// TIA Portal V20 export
FUNCTION_BLOCK "CallGlobal"   // FB48, LAD
TITLE = CallGlobal
// All blocks that provide data to the DB Global.Data are called here. That includes blocks to generate system data as well as blocks that connect handle multiple HMIs.
// stored: IsIECCheckEnabled true, MemoryReserve 100, SetENOAutomatically true
   VAR
      statClockSysMemOld { ExternalWritable := 'False'} : Byte;   // Old value system memory evaluation
      statPulse : Array[0..9] of Bool;
      instLAF_PowerOnOff { ExternalWritable := 'False'} : "LAF_PowerOnOff";
      instLAF_HmiHeaderManager { ExternalWritable := 'False'} : "LAF_HmiHeaderManager";
      instLAF_ClockGen { ExternalWritable := 'False'} : "LAF_ClockGenerator";
      instLSNTP_Server { ExternalWritable := 'False'} : "LSNTP_Server";
      statTonTimer { ExternalWritable := 'False'} : Array[0..9] of TON_TIME;
   END_VAR
   VAR_TEMP
      tempIndex : DInt;   // Temp variable for for loop
      tempAcknowledge : Bool;   // Summarized acknowledge command
      tempPowerOff : Bool;   // Summarized power off command
      tempPowerOn : Bool;   // Summarized power on command
      tempPowerStatus : Int;   // 0 - Off, 1 - Paused, 2 - On
      tempResultXor : Byte;   // Interim result of XOR operation
      tempPosPulse : Byte;   // Interim result puls calculation
      temp_REPLACE_THIS : HW_ANY;
   END_VAR
   VAR CONSTANT
      RESET_BUTTON__COULD_BE_ADDED_HERE : Bool := false;   // Placeholder for a potential global reset button
      TRUE : Bool := TRUE;
      FALSE : Bool := FALSE;
   END_VAR
   VAR_TEMP   // added for the SCL form of the ladder/FBD networks
      _w1 : Bool;
      _w2 : Bool;
      _w3 : Bool;
      _w4 : Bool;
      _w5 : Bool;
      _w6 : Bool;
      _w7 : Bool;
      _w8 : Bool;
   END_VAR
BEGIN

REGION Network 1 (SCL): Summarize HMI commands
   // Read commands for acknowledge, powerOn and powerOff from the different HMI panels and summarize them in temp variables for further logic in this block.
   // Initialize temp variables
   #tempAcknowledge :=
   #tempPowerOff :=
   #tempPowerOn := FALSE;

   // Loop through the HMI panels and summarize the commands
   FOR #tempIndex := 0 TO "NO_OF_PANELS" DO
       #tempAcknowledge := #tempAcknowledge OR "Hmi".mainHeader[#tempIndex].hmiToPlc.acknowledge;
       #tempPowerOff := #tempPowerOff OR "Hmi".mainHeader[#tempIndex].hmiToPlc.powerCommands.%X0;
       #tempPowerOn := #tempPowerOn OR "Hmi".mainHeader[#tempIndex].hmiToPlc.powerCommands.%X1;
   END_FOR;
END_REGION

REGION Network 2: Global Acknowledge
   // The global acknowledge command from the hmi button is assigned to Global.Data.general.acknowledge: This bit it forwarded to all underlaying modules
   // If a hard-wired global reset button exists, it can
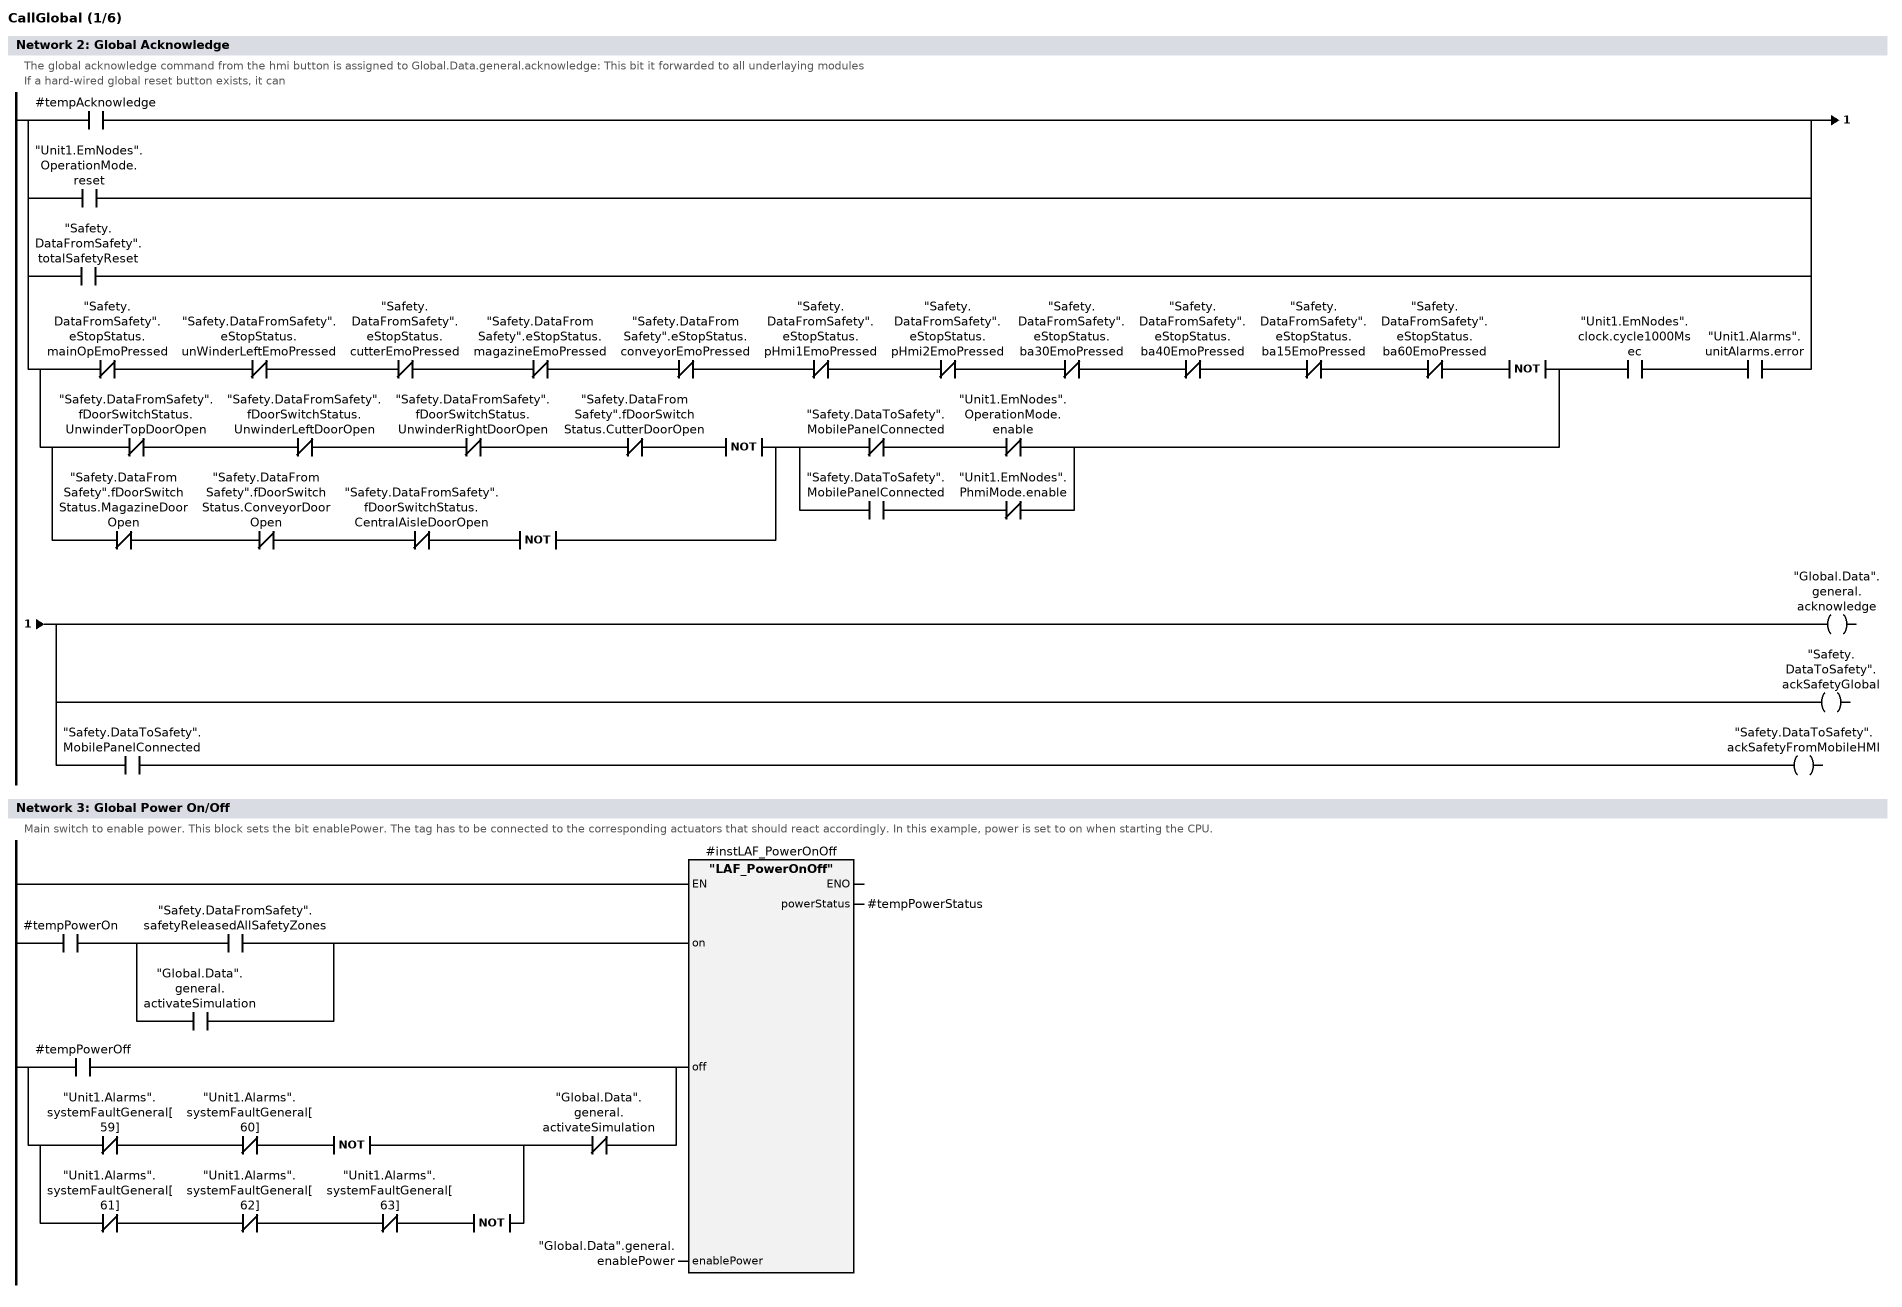
   RUNG wire#powerrail
      Contact( #tempAcknowledge )
      wire#w1
      Coil( "Global.Data".general.acknowledge )
   END_RUNG
   RUNG wire#powerrail
      Contact( "Unit1.EmNodes".OperationMode.reset )
   END_RUNG wire#w1
   RUNG wire#powerrail
      Contact( "Safety.DataFromSafety".totalSafetyReset )
   END_RUNG wire#w1
   RUNG wire#powerrail
      I_Contact( "Safety.DataFromSafety".eStopStatus.mainOpEmoPressed )
      I_Contact( "Safety.DataFromSafety".eStopStatus.unWinderLeftEmoPressed )
      I_Contact( "Safety.DataFromSafety".eStopStatus.cutterEmoPressed )
      I_Contact( "Safety.DataFromSafety".eStopStatus.magazineEmoPressed )
      I_Contact( "Safety.DataFromSafety".eStopStatus.conveyorEmoPressed )
      I_Contact( "Safety.DataFromSafety".eStopStatus.pHmi1EmoPressed )
      I_Contact( "Safety.DataFromSafety".eStopStatus.pHmi2EmoPressed )
      I_Contact( "Safety.DataFromSafety".eStopStatus.ba30EmoPressed )
      I_Contact( "Safety.DataFromSafety".eStopStatus.ba40EmoPressed )
      I_Contact( "Safety.DataFromSafety".eStopStatus.ba15EmoPressed )
      I_Contact( "Safety.DataFromSafety".eStopStatus.ba60EmoPressed )
      Not()
      wire#w2
      Contact( "Unit1.EmNodes".clock.cycle1000Msec )
      Contact( "Unit1.Alarms".unitAlarms.error )
   END_RUNG wire#w1
   RUNG wire#powerrail
      I_Contact( "Safety.DataFromSafety".fDoorSwitchStatus.UnwinderTopDoorOpen )
      I_Contact( "Safety.DataFromSafety".fDoorSwitchStatus.UnwinderLeftDoorOpen )
      I_Contact( "Safety.DataFromSafety".fDoorSwitchStatus.UnwinderRightDoorOpen )
      I_Contact( "Safety.DataFromSafety".fDoorSwitchStatus.CutterDoorOpen )
      Not()
      wire#w3
      I_Contact( "Safety.DataToSafety".MobilePanelConnected )
      I_Contact( "Unit1.EmNodes".OperationMode.enable )
   END_RUNG wire#w2
   RUNG wire#powerrail
      I_Contact( "Safety.DataFromSafety".fDoorSwitchStatus.MagazineDoorOpen )
      I_Contact( "Safety.DataFromSafety".fDoorSwitchStatus.ConveyorDoorOpen )
      I_Contact( "Safety.DataFromSafety".fDoorSwitchStatus.CentralAisleDoorOpen )
      Not()
   END_RUNG wire#w3
   RUNG wire#w3
      Contact( "Safety.DataToSafety".MobilePanelConnected )
      I_Contact( "Unit1.EmNodes".PhmiMode.enable )
   END_RUNG wire#w2
   RUNG wire#w1
      Coil( "Safety.DataToSafety".ackSafetyGlobal )
   END_RUNG
   RUNG wire#w1
      Contact( "Safety.DataToSafety".MobilePanelConnected )
      Coil( "Safety.DataToSafety".ackSafetyFromMobileHMI )
   END_RUNG
   // the same network as SCL:
   "Global.Data".general.acknowledge := #tempAcknowledge OR "Unit1.EmNodes".OperationMode.reset OR "Safety.DataFromSafety".totalSafetyReset OR ((NOT (NOT "Safety.DataFromSafety".eStopStatus.mainOpEmoPressed AND NOT "Safety.DataFromSafety".eStopStatus.unWinderLeftEmoPressed AND NOT "Safety.DataFromSafety".eStopStatus.cutterEmoPressed AND NOT "Safety.DataFromSafety".eStopStatus.magazineEmoPressed AND NOT "Safety.DataFromSafety".eStopStatus.conveyorEmoPressed AND NOT "Safety.DataFromSafety".eStopStatus.pHmi1EmoPressed AND NOT "Safety.DataFromSafety".eStopStatus.pHmi2EmoPressed AND NOT "Safety.DataFromSafety".eStopStatus.ba30EmoPressed AND NOT "Safety.DataFromSafety".eStopStatus.ba40EmoPressed AND NOT "Safety.DataFromSafety".eStopStatus.ba15EmoPressed AND NOT "Safety.DataFromSafety".eStopStatus.ba60EmoPressed) OR ((NOT (NOT "Safety.DataFromSafety".fDoorSwitchStatus.UnwinderTopDoorOpen AND NOT "Safety.DataFromSafety".fDoorSwitchStatus.UnwinderLeftDoorOpen AND NOT "Safety.DataFromSafety".fDoorSwitchStatus.UnwinderRightDoorOpen AND NOT "Safety.DataFromSafety".fDoorSwitchStatus.CutterDoorOpen) OR NOT (NOT "Safety.DataFromSafety".fDoorSwitchStatus.MagazineDoorOpen AND NOT "Safety.DataFromSafety".fDoorSwitchStatus.ConveyorDoorOpen AND NOT "Safety.DataFromSafety".fDoorSwitchStatus.CentralAisleDoorOpen)) AND ((NOT "Safety.DataToSafety".MobilePanelConnected AND NOT "Unit1.EmNodes".OperationMode.enable) OR ("Safety.DataToSafety".MobilePanelConnected AND NOT "Unit1.EmNodes".PhmiMode.enable)))) AND "Unit1.EmNodes".clock.cycle1000Msec AND "Unit1.Alarms".unitAlarms.error);
   "Safety.DataToSafety".ackSafetyGlobal := "Global.Data".general.acknowledge;
   "Safety.DataToSafety".ackSafetyFromMobileHMI := "Global.Data".general.acknowledge AND "Safety.DataToSafety".MobilePanelConnected;
END_REGION

REGION Network 3: Global Power On/Off
   // Main switch to enable power. This block sets the bit enablePower. The tag has to be connected to the corresponding actuators that should react accordingly. In this example, power is set to on when starting the CPU.
   RUNG wire#powerrail
      #instLAF_PowerOnOff(on := wire#w2, off := wire#w4, enablePower := "Global.Data".general.enablePower, powerStatus => #tempPowerStatus)
   END_RUNG
   RUNG wire#powerrail
      Contact( #tempPowerOn )
      wire#w1
      Contact( "Safety.DataFromSafety".safetyReleasedAllSafetyZones )
   END_RUNG wire#w2
   RUNG wire#w1
      Contact( "Global.Data".general.activateSimulation )
   END_RUNG wire#w2
   RUNG wire#powerrail
      Contact( #tempPowerOff )
   END_RUNG wire#w4
   RUNG wire#powerrail
      I_Contact( "Unit1.Alarms".systemFaultGeneral[59] )
      I_Contact( "Unit1.Alarms".systemFaultGeneral[60] )
      Not()
      wire#w3
      I_Contact( "Global.Data".general.activateSimulation )
   END_RUNG wire#w4
   RUNG wire#powerrail
      I_Contact( "Unit1.Alarms".systemFaultGeneral[61] )
      I_Contact( "Unit1.Alarms".systemFaultGeneral[62] )
      I_Contact( "Unit1.Alarms".systemFaultGeneral[63] )
      Not()
   END_RUNG wire#w3
   // the same network as SCL:
   #instLAF_PowerOnOff(on := #tempPowerOn AND ("Safety.DataFromSafety".safetyReleasedAllSafetyZones OR "Global.Data".general.activateSimulation),   // "LAF_PowerOnOff"
                       off := #tempPowerOff OR ((NOT (NOT "Unit1.Alarms".systemFaultGeneral[59] AND NOT "Unit1.Alarms".systemFaultGeneral[60]) OR NOT (NOT "Unit1.Alarms".systemFaultGeneral[61] AND NOT "Unit1.Alarms".systemFaultGeneral[62] AND NOT "Unit1.Alarms".systemFaultGeneral[63])) AND NOT "Global.Data".general.activateSimulation),
                       enablePower := "Global.Data".general.enablePower,
                       powerStatus => #tempPowerStatus);
END_REGION

REGION Network 4 (SCL): Write power status to HMI panels
   // Write power status back to all connected HMI panels
   // Loop through the panels and set the power status
   FOR #tempIndex := 0 TO "NO_OF_PANELS" DO
       "Hmi".mainHeader[#tempIndex].plcToHmi.powerStatus := #tempPowerStatus;
   END_FOR;
END_REGION

REGION Network 5: Special Function Buttons Operator Control Allowed
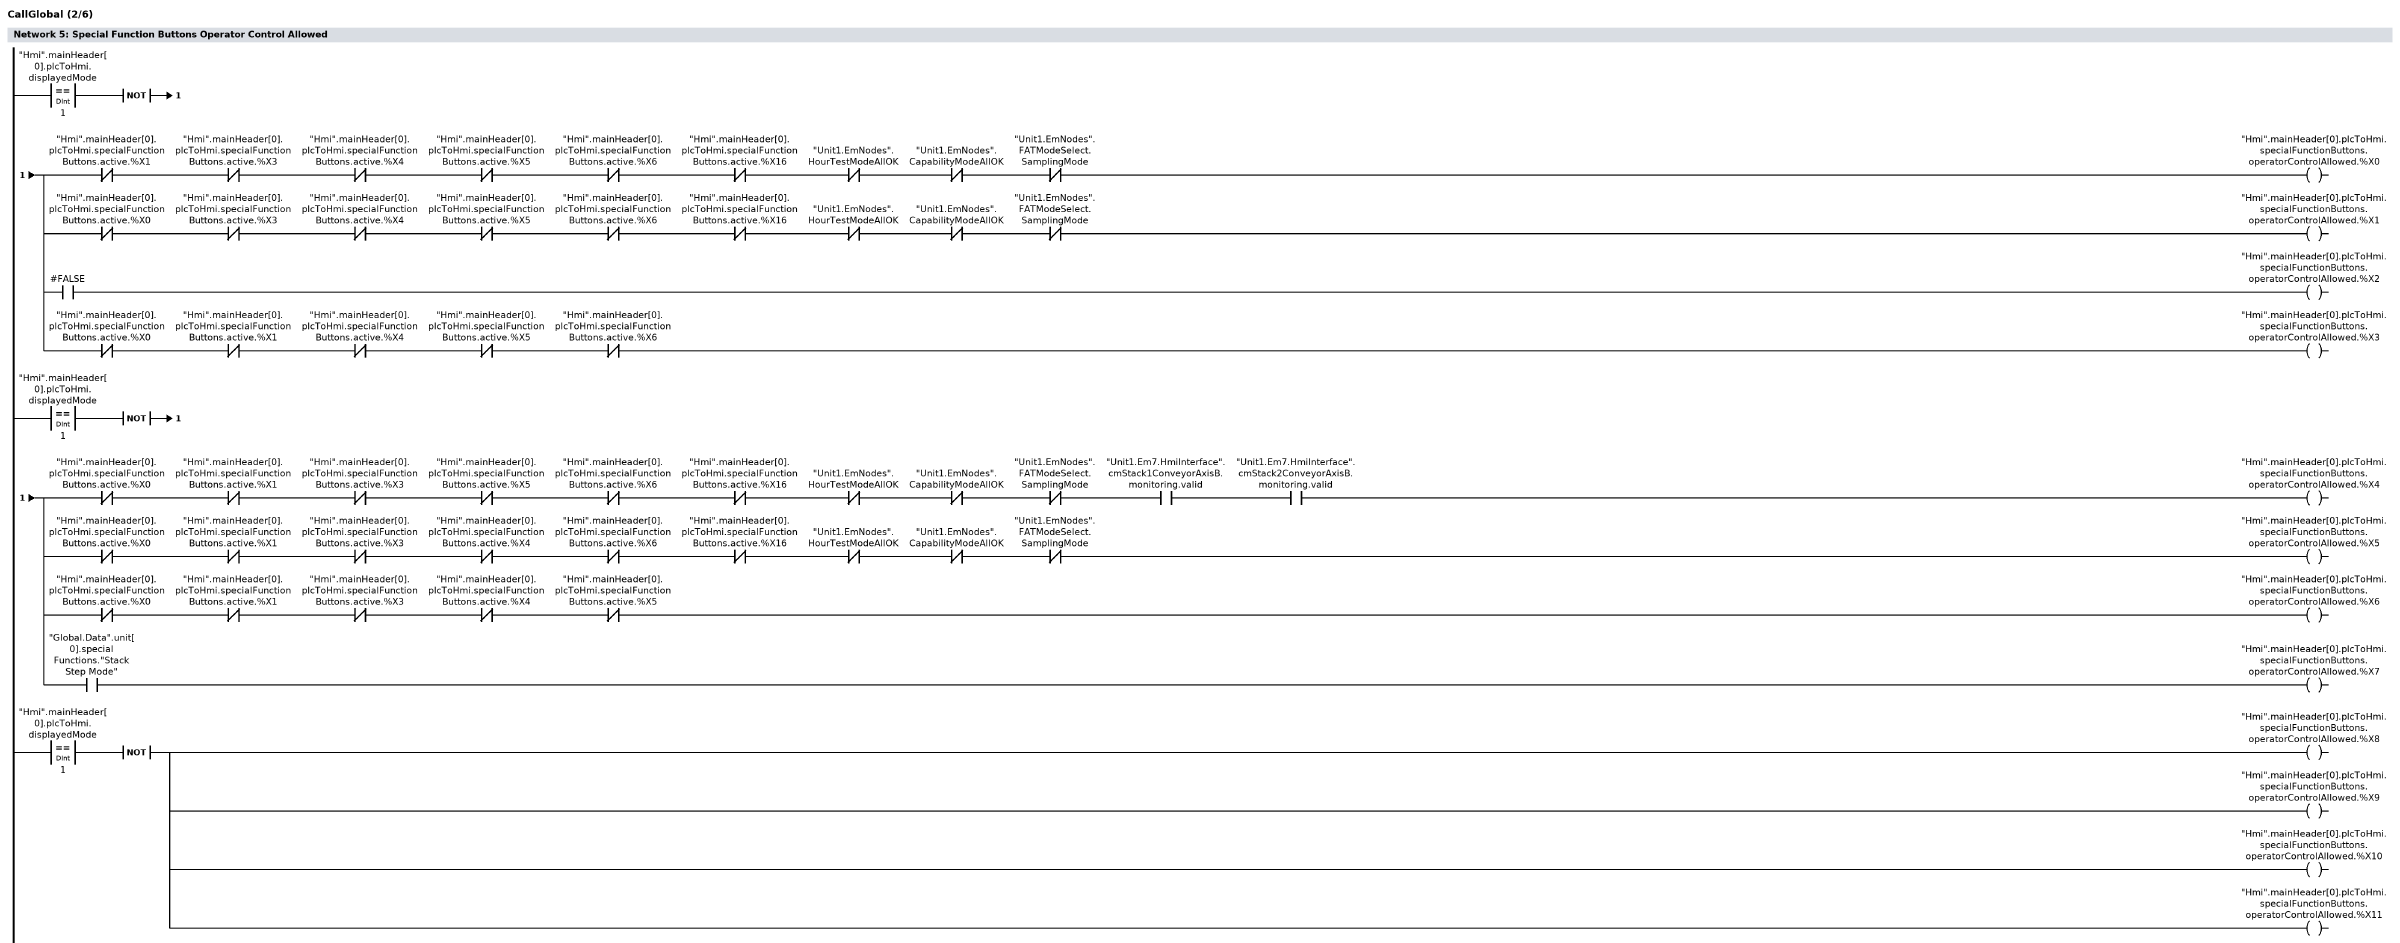
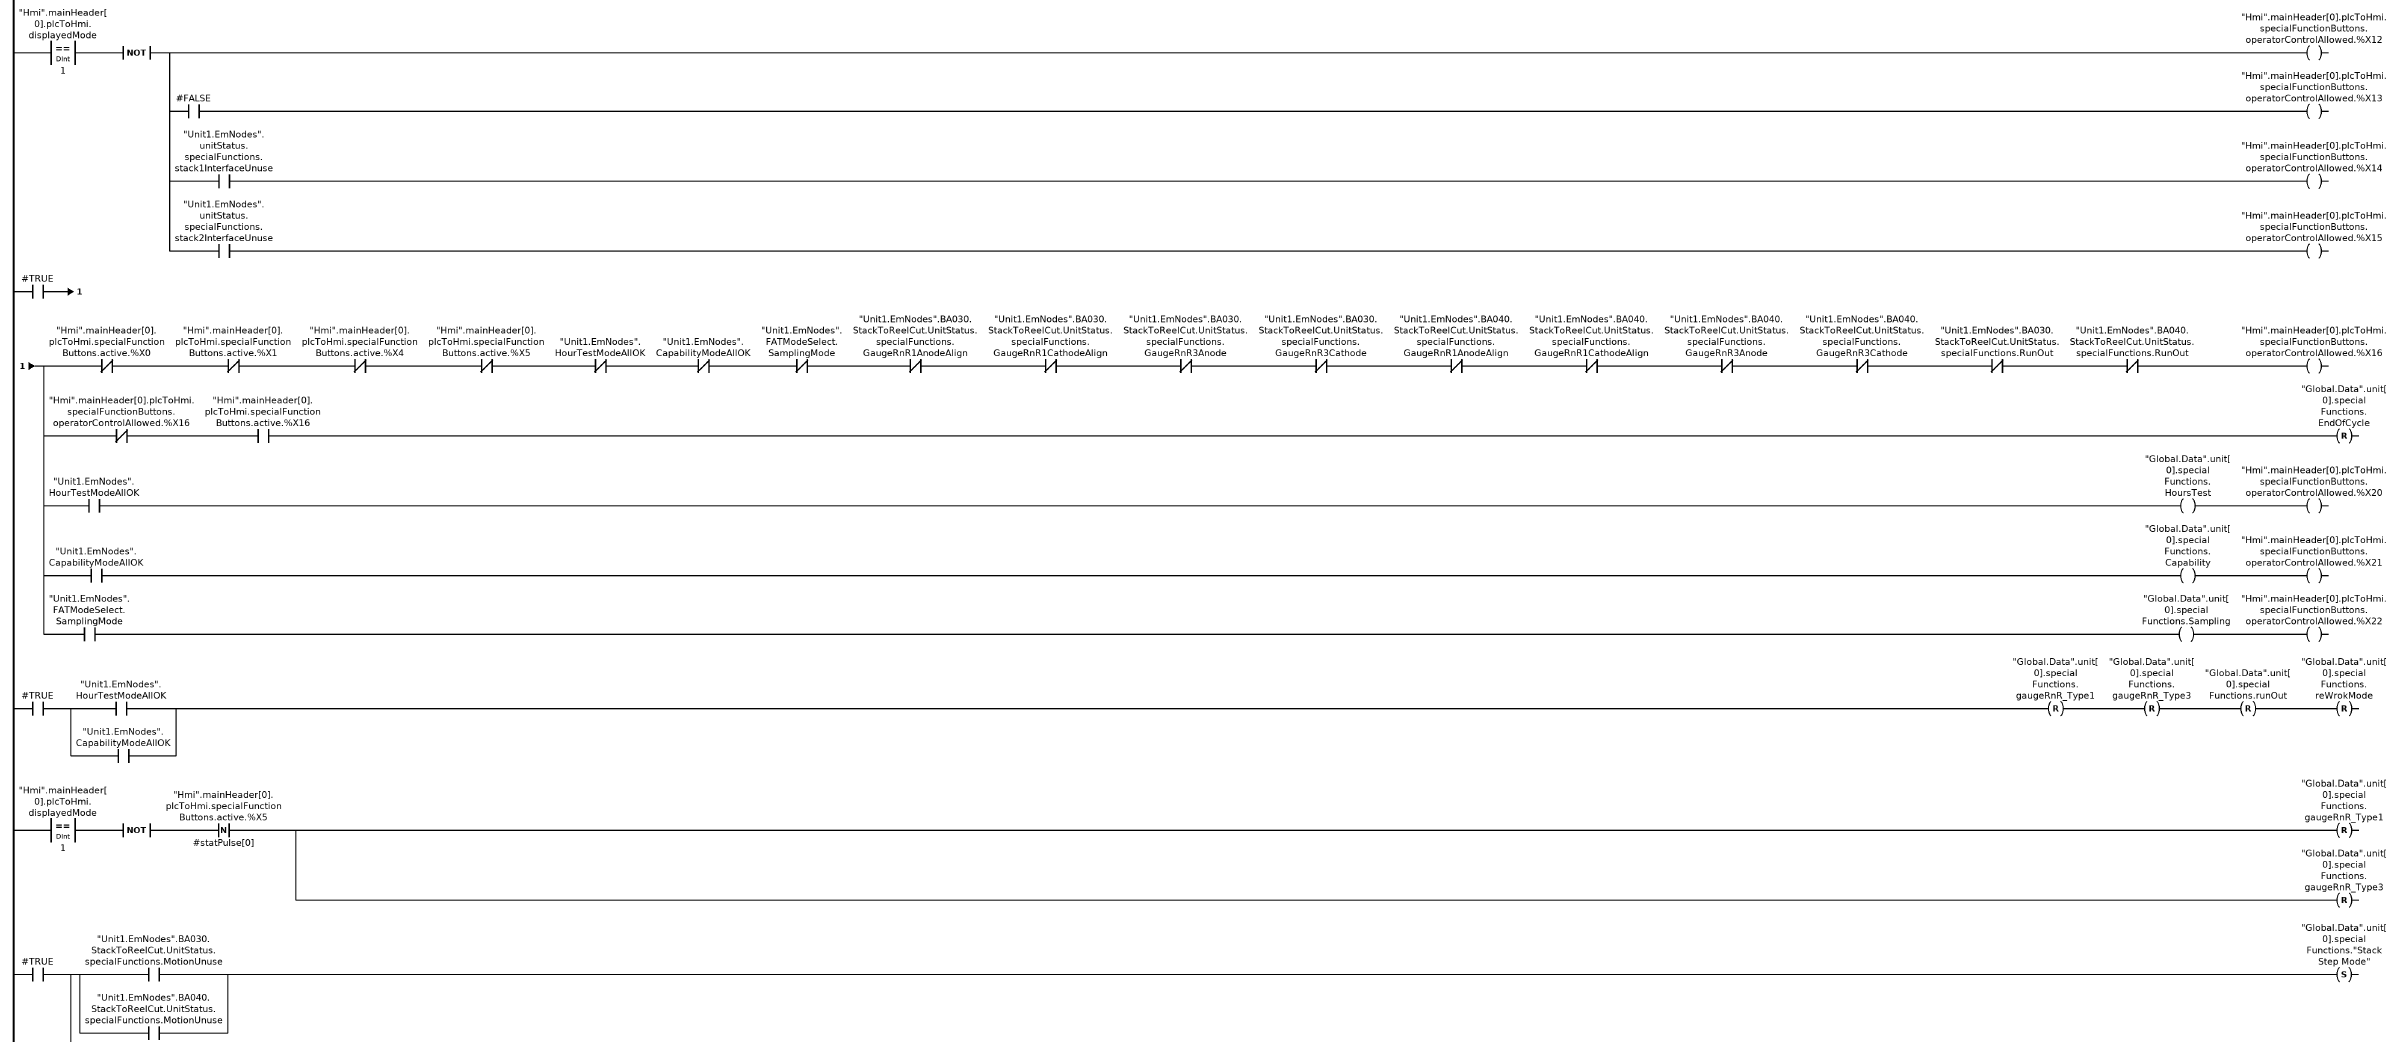
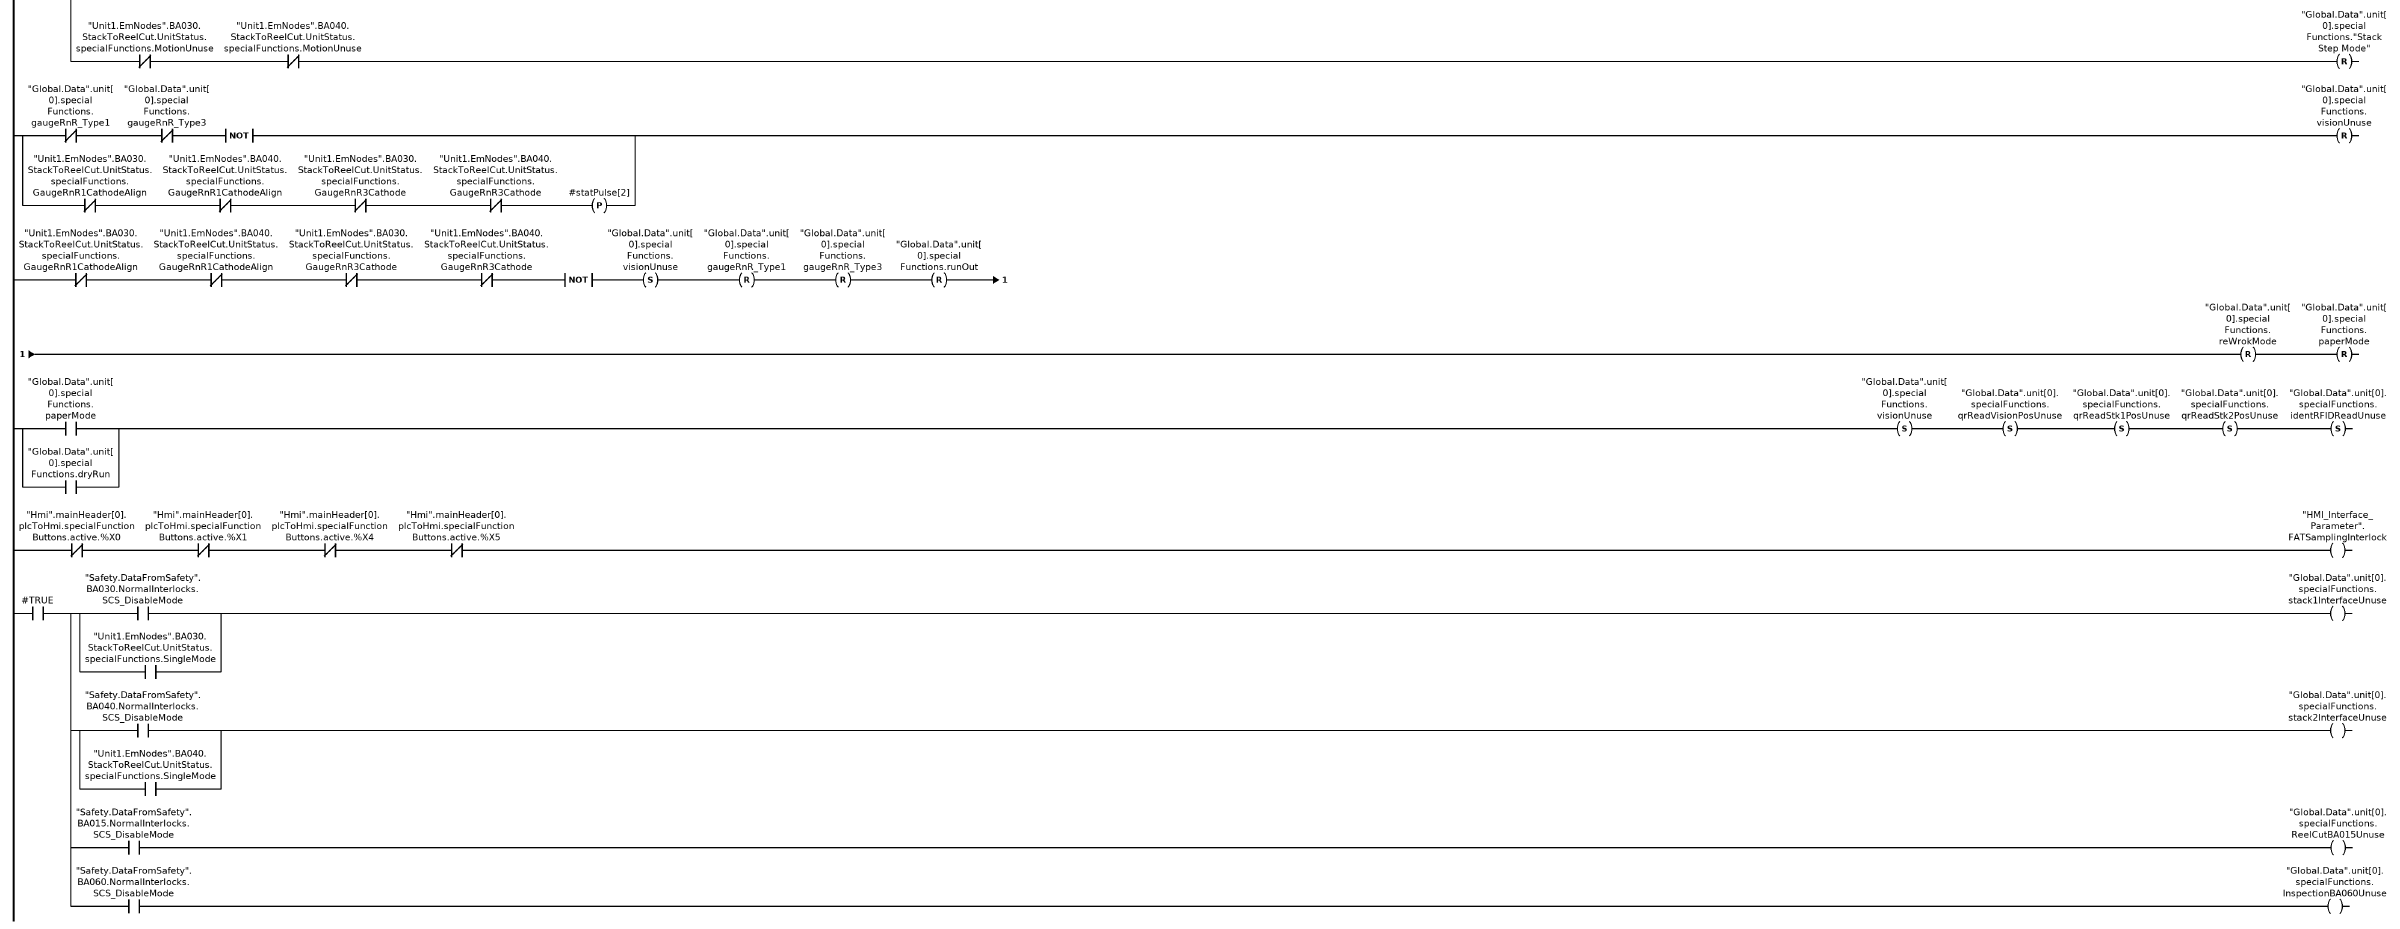
   RUNG wire#powerrail
      { S7_Templates := "SrcType := DInt" } EQ_Contact(in1 := "Hmi".mainHeader[0].plcToHmi.displayedMode, in2 := 1)
      Not()
      wire#w1
      I_Contact( "Hmi".mainHeader[0].plcToHmi.specialFunctionButtons.active.%X1 )
      I_Contact( "Hmi".mainHeader[0].plcToHmi.specialFunctionButtons.active.%X3 )
      I_Contact( "Hmi".mainHeader[0].plcToHmi.specialFunctionButtons.active.%X4 )
      I_Contact( "Hmi".mainHeader[0].plcToHmi.specialFunctionButtons.active.%X5 )
      I_Contact( "Hmi".mainHeader[0].plcToHmi.specialFunctionButtons.active.%X6 )
      I_Contact( "Hmi".mainHeader[0].plcToHmi.specialFunctionButtons.active.%X16 )
      I_Contact( "Unit1.EmNodes".HourTestModeAllOK )
      I_Contact( "Unit1.EmNodes".CapabilityModeAllOK )
      I_Contact( "Unit1.EmNodes".FATModeSelect.SamplingMode )
      Coil( "Hmi".mainHeader[0].plcToHmi.specialFunctionButtons.operatorControlAllowed.%X0 )
   END_RUNG
   RUNG wire#w1
      I_Contact( "Hmi".mainHeader[0].plcToHmi.specialFunctionButtons.active.%X0 )
      I_Contact( "Hmi".mainHeader[0].plcToHmi.specialFunctionButtons.active.%X3 )
      I_Contact( "Hmi".mainHeader[0].plcToHmi.specialFunctionButtons.active.%X4 )
      I_Contact( "Hmi".mainHeader[0].plcToHmi.specialFunctionButtons.active.%X5 )
      I_Contact( "Hmi".mainHeader[0].plcToHmi.specialFunctionButtons.active.%X6 )
      I_Contact( "Hmi".mainHeader[0].plcToHmi.specialFunctionButtons.active.%X16 )
      I_Contact( "Unit1.EmNodes".HourTestModeAllOK )
      I_Contact( "Unit1.EmNodes".CapabilityModeAllOK )
      I_Contact( "Unit1.EmNodes".FATModeSelect.SamplingMode )
      Coil( "Hmi".mainHeader[0].plcToHmi.specialFunctionButtons.operatorControlAllowed.%X1 )
   END_RUNG
   RUNG wire#w1
      Contact( #FALSE )
      Coil( "Hmi".mainHeader[0].plcToHmi.specialFunctionButtons.operatorControlAllowed.%X2 )
   END_RUNG
   RUNG wire#w1
      I_Contact( "Hmi".mainHeader[0].plcToHmi.specialFunctionButtons.active.%X0 )
      I_Contact( "Hmi".mainHeader[0].plcToHmi.specialFunctionButtons.active.%X1 )
      I_Contact( "Hmi".mainHeader[0].plcToHmi.specialFunctionButtons.active.%X4 )
      I_Contact( "Hmi".mainHeader[0].plcToHmi.specialFunctionButtons.active.%X5 )
      I_Contact( "Hmi".mainHeader[0].plcToHmi.specialFunctionButtons.active.%X6 )
      Coil( "Hmi".mainHeader[0].plcToHmi.specialFunctionButtons.operatorControlAllowed.%X3 )
   END_RUNG
   RUNG wire#powerrail
      { S7_Templates := "SrcType := DInt" } EQ_Contact(in1 := "Hmi".mainHeader[0].plcToHmi.displayedMode, in2 := 1)
      Not()
      wire#w2
      I_Contact( "Hmi".mainHeader[0].plcToHmi.specialFunctionButtons.active.%X0 )
      I_Contact( "Hmi".mainHeader[0].plcToHmi.specialFunctionButtons.active.%X1 )
      I_Contact( "Hmi".mainHeader[0].plcToHmi.specialFunctionButtons.active.%X3 )
      I_Contact( "Hmi".mainHeader[0].plcToHmi.specialFunctionButtons.active.%X5 )
      I_Contact( "Hmi".mainHeader[0].plcToHmi.specialFunctionButtons.active.%X6 )
      I_Contact( "Hmi".mainHeader[0].plcToHmi.specialFunctionButtons.active.%X16 )
      I_Contact( "Unit1.EmNodes".HourTestModeAllOK )
      I_Contact( "Unit1.EmNodes".CapabilityModeAllOK )
      I_Contact( "Unit1.EmNodes".FATModeSelect.SamplingMode )
      Contact( "Unit1.Em7.HmiInterface".cmStack1ConveyorAxisB.monitoring.valid )
      Contact( "Unit1.Em7.HmiInterface".cmStack2ConveyorAxisB.monitoring.valid )
      Coil( "Hmi".mainHeader[0].plcToHmi.specialFunctionButtons.operatorControlAllowed.%X4 )
   END_RUNG
   RUNG wire#w2
      I_Contact( "Hmi".mainHeader[0].plcToHmi.specialFunctionButtons.active.%X0 )
      I_Contact( "Hmi".mainHeader[0].plcToHmi.specialFunctionButtons.active.%X1 )
      I_Contact( "Hmi".mainHeader[0].plcToHmi.specialFunctionButtons.active.%X3 )
      I_Contact( "Hmi".mainHeader[0].plcToHmi.specialFunctionButtons.active.%X4 )
      I_Contact( "Hmi".mainHeader[0].plcToHmi.specialFunctionButtons.active.%X6 )
      I_Contact( "Hmi".mainHeader[0].plcToHmi.specialFunctionButtons.active.%X16 )
      I_Contact( "Unit1.EmNodes".HourTestModeAllOK )
      I_Contact( "Unit1.EmNodes".CapabilityModeAllOK )
      I_Contact( "Unit1.EmNodes".FATModeSelect.SamplingMode )
      Coil( "Hmi".mainHeader[0].plcToHmi.specialFunctionButtons.operatorControlAllowed.%X5 )
   END_RUNG
   RUNG wire#w2
      I_Contact( "Hmi".mainHeader[0].plcToHmi.specialFunctionButtons.active.%X0 )
      I_Contact( "Hmi".mainHeader[0].plcToHmi.specialFunctionButtons.active.%X1 )
      I_Contact( "Hmi".mainHeader[0].plcToHmi.specialFunctionButtons.active.%X3 )
      I_Contact( "Hmi".mainHeader[0].plcToHmi.specialFunctionButtons.active.%X4 )
      I_Contact( "Hmi".mainHeader[0].plcToHmi.specialFunctionButtons.active.%X5 )
      Coil( "Hmi".mainHeader[0].plcToHmi.specialFunctionButtons.operatorControlAllowed.%X6 )
   END_RUNG
   RUNG wire#w2
      Contact( "Global.Data".unit[0].specialFunctions."Stack Step Mode" )
      Coil( "Hmi".mainHeader[0].plcToHmi.specialFunctionButtons.operatorControlAllowed.%X7 )
   END_RUNG
   RUNG wire#powerrail
      { S7_Templates := "SrcType := DInt" } EQ_Contact(in1 := "Hmi".mainHeader[0].plcToHmi.displayedMode, in2 := 1)
      Not()
      wire#w3
      Coil( "Hmi".mainHeader[0].plcToHmi.specialFunctionButtons.operatorControlAllowed.%X8 )
   END_RUNG
   RUNG wire#w3
      Coil( "Hmi".mainHeader[0].plcToHmi.specialFunctionButtons.operatorControlAllowed.%X9 )
   END_RUNG
   RUNG wire#w3
      Coil( "Hmi".mainHeader[0].plcToHmi.specialFunctionButtons.operatorControlAllowed.%X10 )
   END_RUNG
   RUNG wire#w3
      Coil( "Hmi".mainHeader[0].plcToHmi.specialFunctionButtons.operatorControlAllowed.%X11 )
   END_RUNG
   RUNG wire#powerrail
      { S7_Templates := "SrcType := DInt" } EQ_Contact(in1 := "Hmi".mainHeader[0].plcToHmi.displayedMode, in2 := 1)
      Not()
      wire#w4
      Coil( "Hmi".mainHeader[0].plcToHmi.specialFunctionButtons.operatorControlAllowed.%X12 )
   END_RUNG
   RUNG wire#w4
      Contact( #FALSE )
      Coil( "Hmi".mainHeader[0].plcToHmi.specialFunctionButtons.operatorControlAllowed.%X13 )
   END_RUNG
   RUNG wire#w4
      Contact( "Unit1.EmNodes".unitStatus.specialFunctions.stack1InterfaceUnuse )
      Coil( "Hmi".mainHeader[0].plcToHmi.specialFunctionButtons.operatorControlAllowed.%X14 )
   END_RUNG
   RUNG wire#w4
      Contact( "Unit1.EmNodes".unitStatus.specialFunctions.stack2InterfaceUnuse )
      Coil( "Hmi".mainHeader[0].plcToHmi.specialFunctionButtons.operatorControlAllowed.%X15 )
   END_RUNG
   RUNG wire#powerrail
      Contact( #TRUE )
      wire#w5
      I_Contact( "Hmi".mainHeader[0].plcToHmi.specialFunctionButtons.active.%X0 )
      I_Contact( "Hmi".mainHeader[0].plcToHmi.specialFunctionButtons.active.%X1 )
      I_Contact( "Hmi".mainHeader[0].plcToHmi.specialFunctionButtons.active.%X4 )
      I_Contact( "Hmi".mainHeader[0].plcToHmi.specialFunctionButtons.active.%X5 )
      I_Contact( "Unit1.EmNodes".HourTestModeAllOK )
      I_Contact( "Unit1.EmNodes".CapabilityModeAllOK )
      I_Contact( "Unit1.EmNodes".FATModeSelect.SamplingMode )
      I_Contact( "Unit1.EmNodes".BA030.StackToReelCut.UnitStatus.specialFunctions.GaugeRnR1AnodeAlign )
      I_Contact( "Unit1.EmNodes".BA030.StackToReelCut.UnitStatus.specialFunctions.GaugeRnR1CathodeAlign )
      I_Contact( "Unit1.EmNodes".BA030.StackToReelCut.UnitStatus.specialFunctions.GaugeRnR3Anode )
      I_Contact( "Unit1.EmNodes".BA030.StackToReelCut.UnitStatus.specialFunctions.GaugeRnR3Cathode )
      I_Contact( "Unit1.EmNodes".BA040.StackToReelCut.UnitStatus.specialFunctions.GaugeRnR1AnodeAlign )
      I_Contact( "Unit1.EmNodes".BA040.StackToReelCut.UnitStatus.specialFunctions.GaugeRnR1CathodeAlign )
      I_Contact( "Unit1.EmNodes".BA040.StackToReelCut.UnitStatus.specialFunctions.GaugeRnR3Anode )
      I_Contact( "Unit1.EmNodes".BA040.StackToReelCut.UnitStatus.specialFunctions.GaugeRnR3Cathode )
      I_Contact( "Unit1.EmNodes".BA030.StackToReelCut.UnitStatus.specialFunctions.RunOut )
      I_Contact( "Unit1.EmNodes".BA040.StackToReelCut.UnitStatus.specialFunctions.RunOut )
      Coil( "Hmi".mainHeader[0].plcToHmi.specialFunctionButtons.operatorControlAllowed.%X16 )
   END_RUNG
   RUNG wire#w5
      I_Contact( "Hmi".mainHeader[0].plcToHmi.specialFunctionButtons.operatorControlAllowed.%X16 )
      Contact( "Hmi".mainHeader[0].plcToHmi.specialFunctionButtons.active.%X16 )
      R_Coil( "Global.Data".unit[0].specialFunctions.EndOfCycle )
   END_RUNG
   RUNG wire#w5
      Contact( "Unit1.EmNodes".HourTestModeAllOK )
      Coil( "Global.Data".unit[0].specialFunctions.HoursTest )
      Coil( "Hmi".mainHeader[0].plcToHmi.specialFunctionButtons.operatorControlAllowed.%X20 )
   END_RUNG
   RUNG wire#w5
      Contact( "Unit1.EmNodes".CapabilityModeAllOK )
      Coil( "Global.Data".unit[0].specialFunctions.Capability )
      Coil( "Hmi".mainHeader[0].plcToHmi.specialFunctionButtons.operatorControlAllowed.%X21 )
   END_RUNG
   RUNG wire#w5
      Contact( "Unit1.EmNodes".FATModeSelect.SamplingMode )
      Coil( "Global.Data".unit[0].specialFunctions.Sampling )
      Coil( "Hmi".mainHeader[0].plcToHmi.specialFunctionButtons.operatorControlAllowed.%X22 )
   END_RUNG
   RUNG wire#powerrail
      Contact( #TRUE )
      wire#w6
      Contact( "Unit1.EmNodes".HourTestModeAllOK )
      wire#w7
      R_Coil( "Global.Data".unit[0].specialFunctions.gaugeRnR_Type1 )
      R_Coil( "Global.Data".unit[0].specialFunctions.gaugeRnR_Type3 )
      R_Coil( "Global.Data".unit[0].specialFunctions.runOut )
      R_Coil( "Global.Data".unit[0].specialFunctions.reWrokMode )
   END_RUNG
   RUNG wire#w6
      Contact( "Unit1.EmNodes".CapabilityModeAllOK )
   END_RUNG wire#w7
   RUNG wire#powerrail
      { S7_Templates := "SrcType := DInt" } EQ_Contact(in1 := "Hmi".mainHeader[0].plcToHmi.displayedMode, in2 := 1)
      Not()
      N_Contact(operand := "Hmi".mainHeader[0].plcToHmi.specialFunctionButtons.active.%X5, bit := #statPulse[0])
      wire#w8
      R_Coil( "Global.Data".unit[0].specialFunctions.gaugeRnR_Type1 )
   END_RUNG
   RUNG wire#w8
      R_Coil( "Global.Data".unit[0].specialFunctions.gaugeRnR_Type3 )
   END_RUNG
   RUNG wire#powerrail
      Contact( #TRUE )
      wire#w9
      Contact( "Unit1.EmNodes".BA030.StackToReelCut.UnitStatus.specialFunctions.MotionUnuse )
      wire#w10
      S_Coil( "Global.Data".unit[0].specialFunctions."Stack Step Mode" )
   END_RUNG
   RUNG wire#w9
      Contact( "Unit1.EmNodes".BA040.StackToReelCut.UnitStatus.specialFunctions.MotionUnuse )
   END_RUNG wire#w10
   RUNG wire#w9
      I_Contact( "Unit1.EmNodes".BA030.StackToReelCut.UnitStatus.specialFunctions.MotionUnuse )
      I_Contact( "Unit1.EmNodes".BA040.StackToReelCut.UnitStatus.specialFunctions.MotionUnuse )
      R_Coil( "Global.Data".unit[0].specialFunctions."Stack Step Mode" )
   END_RUNG
   RUNG wire#powerrail
      I_Contact( "Global.Data".unit[0].specialFunctions.gaugeRnR_Type1 )
      I_Contact( "Global.Data".unit[0].specialFunctions.gaugeRnR_Type3 )
      Not()
      wire#w11
      R_Coil( "Global.Data".unit[0].specialFunctions.visionUnuse )
   END_RUNG
   RUNG wire#powerrail
      I_Contact( "Unit1.EmNodes".BA030.StackToReelCut.UnitStatus.specialFunctions.GaugeRnR1CathodeAlign )
      I_Contact( "Unit1.EmNodes".BA040.StackToReelCut.UnitStatus.specialFunctions.GaugeRnR1CathodeAlign )
      I_Contact( "Unit1.EmNodes".BA030.StackToReelCut.UnitStatus.specialFunctions.GaugeRnR3Cathode )
      I_Contact( "Unit1.EmNodes".BA040.StackToReelCut.UnitStatus.specialFunctions.GaugeRnR3Cathode )
      P_Trig( #statPulse[2] )
   END_RUNG wire#w11
   RUNG wire#powerrail
      I_Contact( "Unit1.EmNodes".BA030.StackToReelCut.UnitStatus.specialFunctions.GaugeRnR1CathodeAlign )
      I_Contact( "Unit1.EmNodes".BA040.StackToReelCut.UnitStatus.specialFunctions.GaugeRnR1CathodeAlign )
      I_Contact( "Unit1.EmNodes".BA030.StackToReelCut.UnitStatus.specialFunctions.GaugeRnR3Cathode )
      I_Contact( "Unit1.EmNodes".BA040.StackToReelCut.UnitStatus.specialFunctions.GaugeRnR3Cathode )
      Not()
      S_Coil( "Global.Data".unit[0].specialFunctions.visionUnuse )
      R_Coil( "Global.Data".unit[0].specialFunctions.gaugeRnR_Type1 )
      R_Coil( "Global.Data".unit[0].specialFunctions.gaugeRnR_Type3 )
      R_Coil( "Global.Data".unit[0].specialFunctions.runOut )
      R_Coil( "Global.Data".unit[0].specialFunctions.reWrokMode )
      R_Coil( "Global.Data".unit[0].specialFunctions.paperMode )
   END_RUNG
   RUNG wire#powerrail
      Contact( "Global.Data".unit[0].specialFunctions.paperMode )
      wire#w12
      S_Coil( "Global.Data".unit[0].specialFunctions.visionUnuse )
      S_Coil( "Global.Data".unit[0].specialFunctions.qrReadVisionPosUnuse )
      S_Coil( "Global.Data".unit[0].specialFunctions.qrReadStk1PosUnuse )
      S_Coil( "Global.Data".unit[0].specialFunctions.qrReadStk2PosUnuse )
      S_Coil( "Global.Data".unit[0].specialFunctions.identRFIDReadUnuse )
   END_RUNG
   RUNG wire#powerrail
      Contact( "Global.Data".unit[0].specialFunctions.dryRun )
   END_RUNG wire#w12
   RUNG wire#powerrail
      I_Contact( "Hmi".mainHeader[0].plcToHmi.specialFunctionButtons.active.%X0 )
      I_Contact( "Hmi".mainHeader[0].plcToHmi.specialFunctionButtons.active.%X1 )
      I_Contact( "Hmi".mainHeader[0].plcToHmi.specialFunctionButtons.active.%X4 )
      I_Contact( "Hmi".mainHeader[0].plcToHmi.specialFunctionButtons.active.%X5 )
      Coil( "HMI_Interface_Parameter".FATSamplingInterlock )
   END_RUNG
   RUNG wire#powerrail
      Contact( #TRUE )
      wire#w13
      Contact( "Safety.DataFromSafety".BA030.NormalInterlocks.SCS_DisableMode )
      wire#w14
      Coil( "Global.Data".unit[0].specialFunctions.stack1InterfaceUnuse )
   END_RUNG
   RUNG wire#w13
      Contact( "Unit1.EmNodes".BA030.StackToReelCut.UnitStatus.specialFunctions.SingleMode )
   END_RUNG wire#w14
   RUNG wire#w13
      Contact( "Safety.DataFromSafety".BA040.NormalInterlocks.SCS_DisableMode )
      wire#w15
      Coil( "Global.Data".unit[0].specialFunctions.stack2InterfaceUnuse )
   END_RUNG
   RUNG wire#w13
      Contact( "Unit1.EmNodes".BA040.StackToReelCut.UnitStatus.specialFunctions.SingleMode )
   END_RUNG wire#w15
   RUNG wire#w13
      Contact( "Safety.DataFromSafety".BA015.NormalInterlocks.SCS_DisableMode )
      Coil( "Global.Data".unit[0].specialFunctions.ReelCutBA015Unuse )
   END_RUNG
   RUNG wire#w13
      Contact( "Safety.DataFromSafety".BA060.NormalInterlocks.SCS_DisableMode )
      Coil( "Global.Data".unit[0].specialFunctions.InspectionBA060Unuse )
   END_RUNG
   // the same network as SCL:
   #_w1 := NOT ("Hmi".mainHeader[0].plcToHmi.displayedMode = 1);
   "Hmi".mainHeader[0].plcToHmi.specialFunctionButtons.operatorControlAllowed.%X0 := #_w1 AND NOT "Hmi".mainHeader[0].plcToHmi.specialFunctionButtons.active.%X1 AND NOT "Hmi".mainHeader[0].plcToHmi.specialFunctionButtons.active.%X3 AND NOT "Hmi".mainHeader[0].plcToHmi.specialFunctionButtons.active.%X4 AND NOT "Hmi".mainHeader[0].plcToHmi.specialFunctionButtons.active.%X5 AND NOT "Hmi".mainHeader[0].plcToHmi.specialFunctionButtons.active.%X6 AND NOT "Hmi".mainHeader[0].plcToHmi.specialFunctionButtons.active.%X16 AND NOT "Unit1.EmNodes".HourTestModeAllOK AND NOT "Unit1.EmNodes".CapabilityModeAllOK AND NOT "Unit1.EmNodes".FATModeSelect.SamplingMode;
   "Hmi".mainHeader[0].plcToHmi.specialFunctionButtons.operatorControlAllowed.%X1 := #_w1 AND NOT "Hmi".mainHeader[0].plcToHmi.specialFunctionButtons.active.%X0 AND NOT "Hmi".mainHeader[0].plcToHmi.specialFunctionButtons.active.%X3 AND NOT "Hmi".mainHeader[0].plcToHmi.specialFunctionButtons.active.%X4 AND NOT "Hmi".mainHeader[0].plcToHmi.specialFunctionButtons.active.%X5 AND NOT "Hmi".mainHeader[0].plcToHmi.specialFunctionButtons.active.%X6 AND NOT "Hmi".mainHeader[0].plcToHmi.specialFunctionButtons.active.%X16 AND NOT "Unit1.EmNodes".HourTestModeAllOK AND NOT "Unit1.EmNodes".CapabilityModeAllOK AND NOT "Unit1.EmNodes".FATModeSelect.SamplingMode;
   "Hmi".mainHeader[0].plcToHmi.specialFunctionButtons.operatorControlAllowed.%X2 := #_w1 AND #FALSE;
   "Hmi".mainHeader[0].plcToHmi.specialFunctionButtons.operatorControlAllowed.%X3 := #_w1 AND NOT "Hmi".mainHeader[0].plcToHmi.specialFunctionButtons.active.%X0 AND NOT "Hmi".mainHeader[0].plcToHmi.specialFunctionButtons.active.%X1 AND NOT "Hmi".mainHeader[0].plcToHmi.specialFunctionButtons.active.%X4 AND NOT "Hmi".mainHeader[0].plcToHmi.specialFunctionButtons.active.%X5 AND NOT "Hmi".mainHeader[0].plcToHmi.specialFunctionButtons.active.%X6;
   #_w2 := NOT ("Hmi".mainHeader[0].plcToHmi.displayedMode = 1);
   "Hmi".mainHeader[0].plcToHmi.specialFunctionButtons.operatorControlAllowed.%X4 := #_w2 AND NOT "Hmi".mainHeader[0].plcToHmi.specialFunctionButtons.active.%X0 AND NOT "Hmi".mainHeader[0].plcToHmi.specialFunctionButtons.active.%X1 AND NOT "Hmi".mainHeader[0].plcToHmi.specialFunctionButtons.active.%X3 AND NOT "Hmi".mainHeader[0].plcToHmi.specialFunctionButtons.active.%X5 AND NOT "Hmi".mainHeader[0].plcToHmi.specialFunctionButtons.active.%X6 AND NOT "Hmi".mainHeader[0].plcToHmi.specialFunctionButtons.active.%X16 AND NOT "Unit1.EmNodes".HourTestModeAllOK AND NOT "Unit1.EmNodes".CapabilityModeAllOK AND NOT "Unit1.EmNodes".FATModeSelect.SamplingMode AND "Unit1.Em7.HmiInterface".cmStack1ConveyorAxisB.monitoring.valid AND "Unit1.Em7.HmiInterface".cmStack2ConveyorAxisB.monitoring.valid;
   "Hmi".mainHeader[0].plcToHmi.specialFunctionButtons.operatorControlAllowed.%X5 := #_w2 AND NOT "Hmi".mainHeader[0].plcToHmi.specialFunctionButtons.active.%X0 AND NOT "Hmi".mainHeader[0].plcToHmi.specialFunctionButtons.active.%X1 AND NOT "Hmi".mainHeader[0].plcToHmi.specialFunctionButtons.active.%X3 AND NOT "Hmi".mainHeader[0].plcToHmi.specialFunctionButtons.active.%X4 AND NOT "Hmi".mainHeader[0].plcToHmi.specialFunctionButtons.active.%X6 AND NOT "Hmi".mainHeader[0].plcToHmi.specialFunctionButtons.active.%X16 AND NOT "Unit1.EmNodes".HourTestModeAllOK AND NOT "Unit1.EmNodes".CapabilityModeAllOK AND NOT "Unit1.EmNodes".FATModeSelect.SamplingMode;
   "Hmi".mainHeader[0].plcToHmi.specialFunctionButtons.operatorControlAllowed.%X6 := #_w2 AND NOT "Hmi".mainHeader[0].plcToHmi.specialFunctionButtons.active.%X0 AND NOT "Hmi".mainHeader[0].plcToHmi.specialFunctionButtons.active.%X1 AND NOT "Hmi".mainHeader[0].plcToHmi.specialFunctionButtons.active.%X3 AND NOT "Hmi".mainHeader[0].plcToHmi.specialFunctionButtons.active.%X4 AND NOT "Hmi".mainHeader[0].plcToHmi.specialFunctionButtons.active.%X5;
   "Hmi".mainHeader[0].plcToHmi.specialFunctionButtons.operatorControlAllowed.%X7 := #_w2 AND "Global.Data".unit[0].specialFunctions."Stack Step Mode";
   #_w3 := NOT ("Hmi".mainHeader[0].plcToHmi.displayedMode = 1);
   "Hmi".mainHeader[0].plcToHmi.specialFunctionButtons.operatorControlAllowed.%X8 := NOT ("Hmi".mainHeader[0].plcToHmi.displayedMode = 1);
   "Hmi".mainHeader[0].plcToHmi.specialFunctionButtons.operatorControlAllowed.%X9 := #_w3;
   "Hmi".mainHeader[0].plcToHmi.specialFunctionButtons.operatorControlAllowed.%X10 := #_w3;
   "Hmi".mainHeader[0].plcToHmi.specialFunctionButtons.operatorControlAllowed.%X11 := #_w3;
   #_w4 := NOT ("Hmi".mainHeader[0].plcToHmi.displayedMode = 1);
   "Hmi".mainHeader[0].plcToHmi.specialFunctionButtons.operatorControlAllowed.%X12 := NOT ("Hmi".mainHeader[0].plcToHmi.displayedMode = 1);
   "Hmi".mainHeader[0].plcToHmi.specialFunctionButtons.operatorControlAllowed.%X13 := #_w4 AND #FALSE;
   "Hmi".mainHeader[0].plcToHmi.specialFunctionButtons.operatorControlAllowed.%X14 := #_w4 AND "Unit1.EmNodes".unitStatus.specialFunctions.stack1InterfaceUnuse;
   "Hmi".mainHeader[0].plcToHmi.specialFunctionButtons.operatorControlAllowed.%X15 := #_w4 AND "Unit1.EmNodes".unitStatus.specialFunctions.stack2InterfaceUnuse;
   "Hmi".mainHeader[0].plcToHmi.specialFunctionButtons.operatorControlAllowed.%X16 := #TRUE AND NOT "Hmi".mainHeader[0].plcToHmi.specialFunctionButtons.active.%X0 AND NOT "Hmi".mainHeader[0].plcToHmi.specialFunctionButtons.active.%X1 AND NOT "Hmi".mainHeader[0].plcToHmi.specialFunctionButtons.active.%X4 AND NOT "Hmi".mainHeader[0].plcToHmi.specialFunctionButtons.active.%X5 AND NOT "Unit1.EmNodes".HourTestModeAllOK AND NOT "Unit1.EmNodes".CapabilityModeAllOK AND NOT "Unit1.EmNodes".FATModeSelect.SamplingMode AND NOT "Unit1.EmNodes".BA030.StackToReelCut.UnitStatus.specialFunctions.GaugeRnR1AnodeAlign AND NOT "Unit1.EmNodes".BA030.StackToReelCut.UnitStatus.specialFunctions.GaugeRnR1CathodeAlign AND NOT "Unit1.EmNodes".BA030.StackToReelCut.UnitStatus.specialFunctions.GaugeRnR3Anode AND NOT "Unit1.EmNodes".BA030.StackToReelCut.UnitStatus.specialFunctions.GaugeRnR3Cathode AND NOT "Unit1.EmNodes".BA040.StackToReelCut.UnitStatus.specialFunctions.GaugeRnR1AnodeAlign AND NOT "Unit1.EmNodes".BA040.StackToReelCut.UnitStatus.specialFunctions.GaugeRnR1CathodeAlign AND NOT "Unit1.EmNodes".BA040.StackToReelCut.UnitStatus.specialFunctions.GaugeRnR3Anode AND NOT "Unit1.EmNodes".BA040.StackToReelCut.UnitStatus.specialFunctions.GaugeRnR3Cathode AND NOT "Unit1.EmNodes".BA030.StackToReelCut.UnitStatus.specialFunctions.RunOut AND NOT "Unit1.EmNodes".BA040.StackToReelCut.UnitStatus.specialFunctions.RunOut;
   IF #TRUE AND NOT "Hmi".mainHeader[0].plcToHmi.specialFunctionButtons.operatorControlAllowed.%X16 AND "Hmi".mainHeader[0].plcToHmi.specialFunctionButtons.active.%X16 THEN
       "Global.Data".unit[0].specialFunctions.EndOfCycle := FALSE;
   END_IF;
   "Global.Data".unit[0].specialFunctions.HoursTest := #TRUE AND "Unit1.EmNodes".HourTestModeAllOK;
   "Hmi".mainHeader[0].plcToHmi.specialFunctionButtons.operatorControlAllowed.%X20 := #TRUE AND "Unit1.EmNodes".HourTestModeAllOK;
   "Global.Data".unit[0].specialFunctions.Capability := #TRUE AND "Unit1.EmNodes".CapabilityModeAllOK;
   "Hmi".mainHeader[0].plcToHmi.specialFunctionButtons.operatorControlAllowed.%X21 := #TRUE AND "Unit1.EmNodes".CapabilityModeAllOK;
   "Global.Data".unit[0].specialFunctions.Sampling := #TRUE AND "Unit1.EmNodes".FATModeSelect.SamplingMode;
   "Hmi".mainHeader[0].plcToHmi.specialFunctionButtons.operatorControlAllowed.%X22 := #TRUE AND "Unit1.EmNodes".FATModeSelect.SamplingMode;
   IF #TRUE AND ("Unit1.EmNodes".HourTestModeAllOK OR "Unit1.EmNodes".CapabilityModeAllOK) THEN
       "Global.Data".unit[0].specialFunctions.gaugeRnR_Type1 := FALSE;
       "Global.Data".unit[0].specialFunctions.gaugeRnR_Type3 := FALSE;
       "Global.Data".unit[0].specialFunctions.runOut := FALSE;
       "Global.Data".unit[0].specialFunctions.reWrokMode := FALSE;
   END_IF;
   #_w5 := NOT ("Hmi".mainHeader[0].plcToHmi.displayedMode = 1) AND NOT "Hmi".mainHeader[0].plcToHmi.specialFunctionButtons.active.%X5 AND #statPulse[0];   // falling edge of "Hmi".mainHeader[0].plcToHmi.specialFunctionButtons.active.%X5
   #statPulse[0] := "Hmi".mainHeader[0].plcToHmi.specialFunctionButtons.active.%X5;
   IF #_w5 THEN
       "Global.Data".unit[0].specialFunctions.gaugeRnR_Type1 := FALSE;
       "Global.Data".unit[0].specialFunctions.gaugeRnR_Type3 := FALSE;
   END_IF;
   IF #TRUE AND ("Unit1.EmNodes".BA030.StackToReelCut.UnitStatus.specialFunctions.MotionUnuse OR "Unit1.EmNodes".BA040.StackToReelCut.UnitStatus.specialFunctions.MotionUnuse) THEN
       "Global.Data".unit[0].specialFunctions."Stack Step Mode" := TRUE;
   END_IF;
   IF #TRUE AND NOT "Unit1.EmNodes".BA030.StackToReelCut.UnitStatus.specialFunctions.MotionUnuse AND NOT "Unit1.EmNodes".BA040.StackToReelCut.UnitStatus.specialFunctions.MotionUnuse THEN
       "Global.Data".unit[0].specialFunctions."Stack Step Mode" := FALSE;
   END_IF;
   #_w6 := NOT "Unit1.EmNodes".BA030.StackToReelCut.UnitStatus.specialFunctions.GaugeRnR1CathodeAlign AND NOT "Unit1.EmNodes".BA040.StackToReelCut.UnitStatus.specialFunctions.GaugeRnR1CathodeAlign AND NOT "Unit1.EmNodes".BA030.StackToReelCut.UnitStatus.specialFunctions.GaugeRnR3Cathode AND NOT "Unit1.EmNodes".BA040.StackToReelCut.UnitStatus.specialFunctions.GaugeRnR3Cathode;
   #_w7 := #_w6 AND NOT #statPulse[2];   // rising edge
   #statPulse[2] := #_w6;
   IF NOT (NOT "Global.Data".unit[0].specialFunctions.gaugeRnR_Type1 AND NOT "Global.Data".unit[0].specialFunctions.gaugeRnR_Type3) OR #_w7 THEN
       "Global.Data".unit[0].specialFunctions.visionUnuse := FALSE;
   END_IF;
   IF NOT (NOT "Unit1.EmNodes".BA030.StackToReelCut.UnitStatus.specialFunctions.GaugeRnR1CathodeAlign AND NOT "Unit1.EmNodes".BA040.StackToReelCut.UnitStatus.specialFunctions.GaugeRnR1CathodeAlign AND NOT "Unit1.EmNodes".BA030.StackToReelCut.UnitStatus.specialFunctions.GaugeRnR3Cathode AND NOT "Unit1.EmNodes".BA040.StackToReelCut.UnitStatus.specialFunctions.GaugeRnR3Cathode) THEN
       "Global.Data".unit[0].specialFunctions.visionUnuse := TRUE;
       "Global.Data".unit[0].specialFunctions.gaugeRnR_Type1 := FALSE;
       "Global.Data".unit[0].specialFunctions.gaugeRnR_Type3 := FALSE;
       "Global.Data".unit[0].specialFunctions.runOut := FALSE;
       "Global.Data".unit[0].specialFunctions.reWrokMode := FALSE;
       "Global.Data".unit[0].specialFunctions.paperMode := FALSE;
   END_IF;
   #_w8 := "Global.Data".unit[0].specialFunctions.paperMode OR "Global.Data".unit[0].specialFunctions.dryRun;
   IF #_w8 THEN
       "Global.Data".unit[0].specialFunctions.visionUnuse := TRUE;
       "Global.Data".unit[0].specialFunctions.qrReadVisionPosUnuse := TRUE;
       "Global.Data".unit[0].specialFunctions.qrReadStk1PosUnuse := TRUE;
       "Global.Data".unit[0].specialFunctions.qrReadStk2PosUnuse := TRUE;
       "Global.Data".unit[0].specialFunctions.identRFIDReadUnuse := TRUE;
   END_IF;
   "HMI_Interface_Parameter".FATSamplingInterlock := NOT "Hmi".mainHeader[0].plcToHmi.specialFunctionButtons.active.%X0 AND NOT "Hmi".mainHeader[0].plcToHmi.specialFunctionButtons.active.%X1 AND NOT "Hmi".mainHeader[0].plcToHmi.specialFunctionButtons.active.%X4 AND NOT "Hmi".mainHeader[0].plcToHmi.specialFunctionButtons.active.%X5;
   "Global.Data".unit[0].specialFunctions.stack1InterfaceUnuse := #TRUE AND ("Safety.DataFromSafety".BA030.NormalInterlocks.SCS_DisableMode OR "Unit1.EmNodes".BA030.StackToReelCut.UnitStatus.specialFunctions.SingleMode);
   "Global.Data".unit[0].specialFunctions.stack2InterfaceUnuse := #TRUE AND ("Safety.DataFromSafety".BA040.NormalInterlocks.SCS_DisableMode OR "Unit1.EmNodes".BA040.StackToReelCut.UnitStatus.specialFunctions.SingleMode);
   "Global.Data".unit[0].specialFunctions.ReelCutBA015Unuse := #TRUE AND "Safety.DataFromSafety".BA015.NormalInterlocks.SCS_DisableMode;
   "Global.Data".unit[0].specialFunctions.InspectionBA060Unuse := #TRUE AND "Safety.DataFromSafety".BA060.NormalInterlocks.SCS_DisableMode;
END_REGION

REGION Network 6: HMI Control Header
   // Read the input from the control header in the HMI an distribute information to the according units. Vice versa, summarize the unit information and provide it to the control header to display e.g. the modes and states.
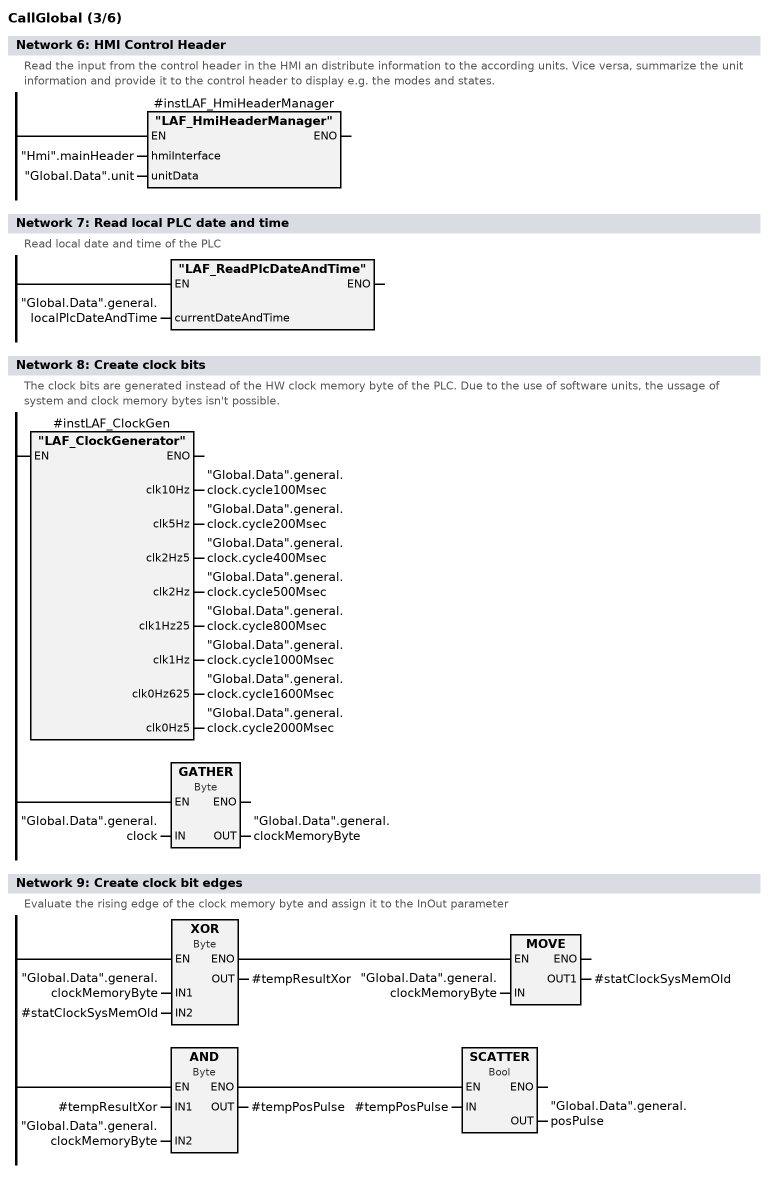
   RUNG wire#powerrail
      #instLAF_HmiHeaderManager(hmiInterface := "Hmi".mainHeader, unitData := "Global.Data".unit)
   END_RUNG
   // the same network as SCL:
   #instLAF_HmiHeaderManager(hmiInterface := "Hmi".mainHeader, unitData := "Global.Data".unit);   // "LAF_HmiHeaderManager"
END_REGION

REGION Network 7: Read local PLC date and time
   // Read local date and time of the PLC
   RUNG wire#powerrail
      "LAF_ReadPlcDateAndTime"(currentDateAndTime := "Global.Data".general.localPlcDateAndTime)
   END_RUNG
   // the same network as SCL:
   "LAF_ReadPlcDateAndTime"(currentDateAndTime := "Global.Data".general.localPlcDateAndTime);
END_REGION

REGION Network 8: Create clock bits
   // The clock bits are generated instead of the HW clock memory byte of the PLC. Due to the use of software units, the ussage of system and clock memory bytes isn't possible.
   RUNG wire#powerrail
      #instLAF_ClockGen(clk10Hz => "Global.Data".general.clock.cycle100Msec, clk5Hz => "Global.Data".general.clock.cycle200Msec, clk2Hz5 => "Global.Data".general.clock.cycle400Msec, clk2Hz => "Global.Data".general.clock.cycle500Msec, clk1Hz25 => "Global.Data".general.clock.cycle800Msec, clk1Hz => "Global.Data".general.clock.cycle1000Msec, clk0Hz625 => "Global.Data".general.clock.cycle1600Msec, clk0Hz5 => "Global.Data".general.clock.cycle2000Msec)
   END_RUNG
   RUNG wire#powerrail
      { S7_Templates := "[dest_type := Byte, src_type := Bool]" } GATHER(IN := "Global.Data".general.clock, OUT => "Global.Data".general.clockMemoryByte)
   END_RUNG
   // the same network as SCL:
   #instLAF_ClockGen(clk10Hz => "Global.Data".general.clock.cycle100Msec,   // "LAF_ClockGenerator"
                     clk5Hz => "Global.Data".general.clock.cycle200Msec,
                     clk2Hz5 => "Global.Data".general.clock.cycle400Msec,
                     clk2Hz => "Global.Data".general.clock.cycle500Msec,
                     clk1Hz25 => "Global.Data".general.clock.cycle800Msec,
                     clk1Hz => "Global.Data".general.clock.cycle1000Msec,
                     clk0Hz625 => "Global.Data".general.clock.cycle1600Msec,
                     clk0Hz5 => "Global.Data".general.clock.cycle2000Msec);
   GATHER(IN := "Global.Data".general.clock, OUT => "Global.Data".general.clockMemoryByte);
END_REGION

REGION Network 9: Create clock bit edges
   // Evaluate the rising edge of the clock memory byte and assign it to the InOut parameter
   #tempResultXor := "Global.Data".general.clockMemoryByte XOR #statClockSysMemOld;
   #statClockSysMemOld := "Global.Data".general.clockMemoryByte;
   #tempPosPulse := #tempResultXor AND "Global.Data".general.clockMemoryByte;
   SCATTER(IN := #tempPosPulse, OUT => "Global.Data".general.posPulse);
END_REGION

REGION Network 10: Time Synchronisation (NTP)
   // With the LSNTP_Server block, the NTP server will be enabled on S7 PLC, to wich the NTP client (e.g. Panel), can synchronize their data and time.
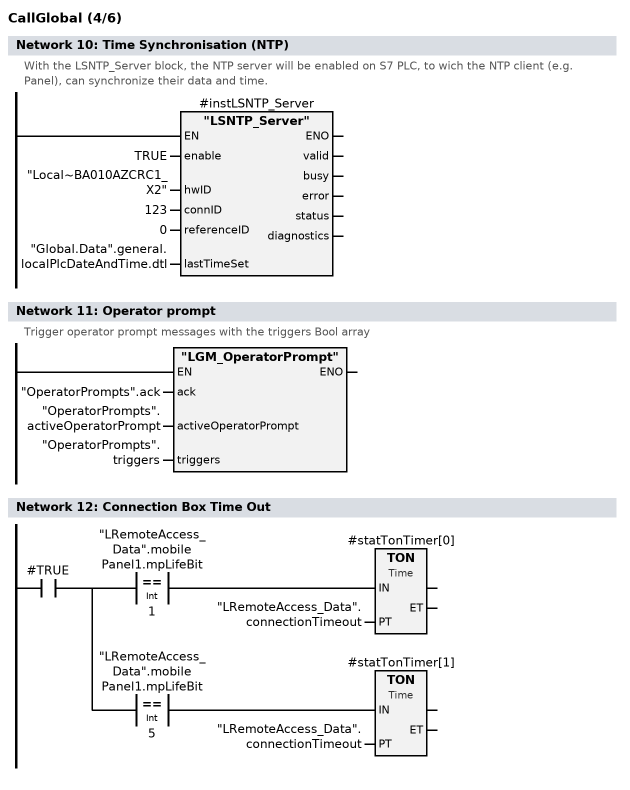
   RUNG wire#powerrail
      #instLSNTP_Server(enable := TRUE, hwID := "Local~BA010AZCRC1_X2", connID := 123, referenceID := 0, lastTimeSet := "Global.Data".general.localPlcDateAndTime.dtl, valid =>, busy =>, error =>, status =>, diagnostics =>)
   END_RUNG
   // the same network as SCL:
   #instLSNTP_Server(enable := TRUE,   // "LSNTP_Server"
                     hwID := "Local~BA010AZCRC1_X2",
                     connID := 123,
                     referenceID := 0,
                     lastTimeSet := "Global.Data".general.localPlcDateAndTime.dtl);
END_REGION

REGION Network 11: Operator prompt
   // Trigger operator prompt messages with the triggers Bool array
   RUNG wire#powerrail
      "LGM_OperatorPrompt"(ack := "OperatorPrompts".ack, activeOperatorPrompt := "OperatorPrompts".activeOperatorPrompt, triggers := "OperatorPrompts".triggers)
   END_RUNG
   // the same network as SCL:
   "LGM_OperatorPrompt"(ack := "OperatorPrompts".ack,
                        activeOperatorPrompt := "OperatorPrompts".activeOperatorPrompt,
                        triggers := "OperatorPrompts".triggers);
END_REGION

REGION Network 12: Connection Box Time Out
   RUNG wire#powerrail
      Contact( #TRUE )
      wire#w1
      { S7_Templates := "SrcType := Int" } EQ_Contact(in1 := "LRemoteAccess_Data".mobilePanel1.mpLifeBit, in2 := 1)
      { S7_Templates := "time_type := Time" } #statTonTimer[0].TON(pt := "LRemoteAccess_Data".connectionTimeout, et =>)
   END_RUNG
   RUNG wire#w1
      { S7_Templates := "SrcType := Int" } EQ_Contact(in1 := "LRemoteAccess_Data".mobilePanel1.mpLifeBit, in2 := 5)
      { S7_Templates := "time_type := Time" } #statTonTimer[1].TON(pt := "LRemoteAccess_Data".connectionTimeout, et =>)
   END_RUNG
   // the same network as SCL:
   #statTonTimer[0].TON(IN := #TRUE AND ("LRemoteAccess_Data".mobilePanel1.mpLifeBit = 1),
                        PT := "LRemoteAccess_Data".connectionTimeout);
   #statTonTimer[1].TON(IN := #TRUE AND ("LRemoteAccess_Data".mobilePanel1.mpLifeBit = 5),
                        PT := "LRemoteAccess_Data".connectionTimeout);
END_REGION

REGION Network 13: Connection box is connected
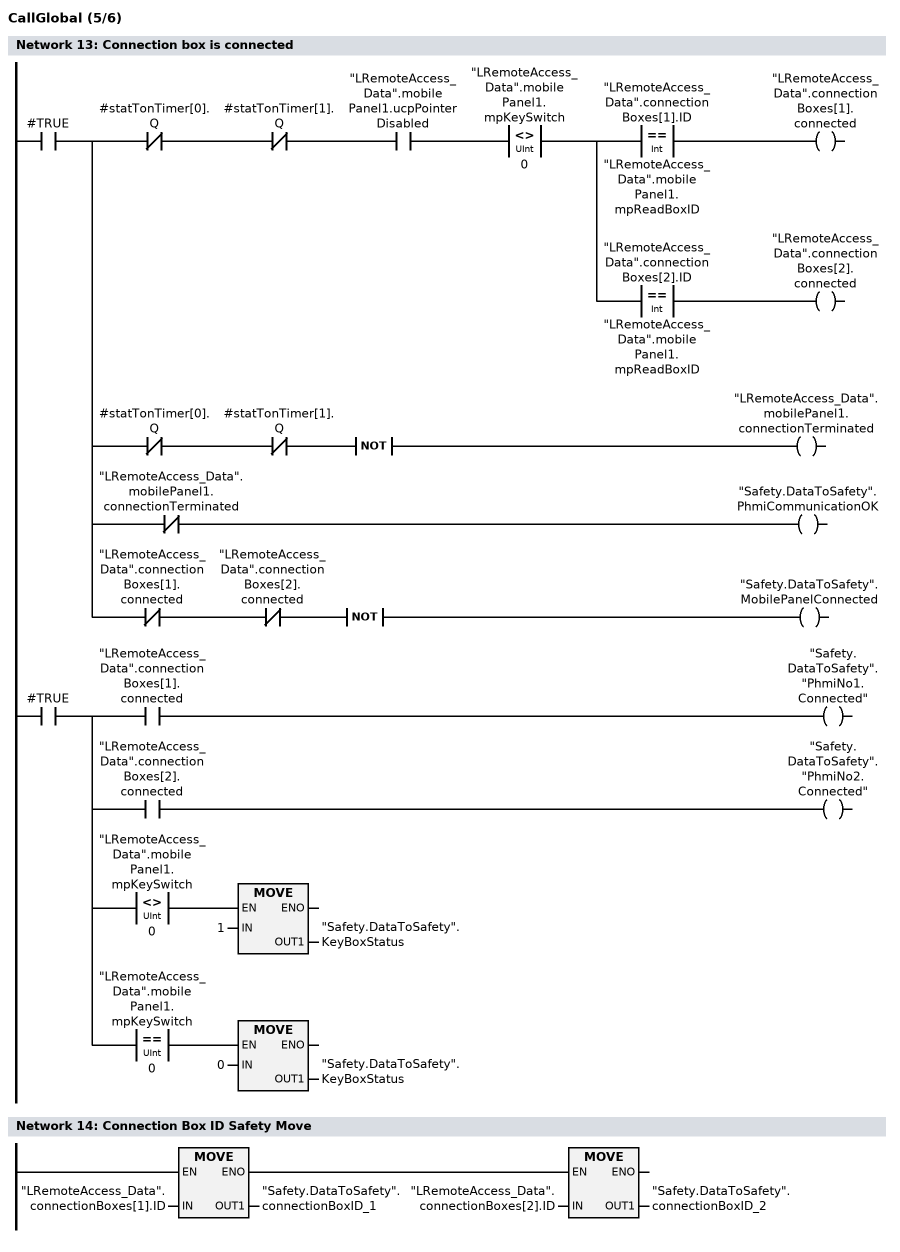
   RUNG wire#powerrail
      Contact( #TRUE )
      wire#w1
      I_Contact( #statTonTimer[0].Q )
      I_Contact( #statTonTimer[1].Q )
      Contact( "LRemoteAccess_Data".mobilePanel1.ucpPointerDisabled )
      { S7_Templates := "SrcType := UInt" } NE_Contact(in1 := "LRemoteAccess_Data".mobilePanel1.mpKeySwitch, in2 := 0)
      wire#w2
      { S7_Templates := "SrcType := Int" } EQ_Contact(in1 := "LRemoteAccess_Data".connectionBoxes[1].ID, in2 := "LRemoteAccess_Data".mobilePanel1.mpReadBoxID)
      Coil( "LRemoteAccess_Data".connectionBoxes[1].connected )
   END_RUNG
   RUNG wire#w2
      { S7_Templates := "SrcType := Int" } EQ_Contact(in1 := "LRemoteAccess_Data".connectionBoxes[2].ID, in2 := "LRemoteAccess_Data".mobilePanel1.mpReadBoxID)
      Coil( "LRemoteAccess_Data".connectionBoxes[2].connected )
   END_RUNG
   RUNG wire#w1
      I_Contact( #statTonTimer[0].Q )
      I_Contact( #statTonTimer[1].Q )
      Not()
      Coil( "LRemoteAccess_Data".mobilePanel1.connectionTerminated )
   END_RUNG
   RUNG wire#w1
      I_Contact( "LRemoteAccess_Data".mobilePanel1.connectionTerminated )
      Coil( "Safety.DataToSafety".PhmiCommunicationOK )
   END_RUNG
   RUNG wire#w1
      I_Contact( "LRemoteAccess_Data".connectionBoxes[1].connected )
      I_Contact( "LRemoteAccess_Data".connectionBoxes[2].connected )
      Not()
      Coil( "Safety.DataToSafety".MobilePanelConnected )
   END_RUNG
   RUNG wire#powerrail
      Contact( #TRUE )
      wire#w3
      Contact( "LRemoteAccess_Data".connectionBoxes[1].connected )
      Coil( "Safety.DataToSafety"."PhmiNo1.Connected" )
   END_RUNG
   RUNG wire#w3
      Contact( "LRemoteAccess_Data".connectionBoxes[2].connected )
      Coil( "Safety.DataToSafety"."PhmiNo2.Connected" )
   END_RUNG
   RUNG wire#w3
      { S7_Templates := "SrcType := UInt" } NE_Contact(in1 := "LRemoteAccess_Data".mobilePanel1.mpKeySwitch, in2 := 0)
      Move(in := 1, out1 => "Safety.DataToSafety".KeyBoxStatus)
   END_RUNG
   RUNG wire#w3
      { S7_Templates := "SrcType := UInt" } EQ_Contact(in1 := "LRemoteAccess_Data".mobilePanel1.mpKeySwitch, in2 := 0)
      Move(in := 0, out1 => "Safety.DataToSafety".KeyBoxStatus)
   END_RUNG
   // the same network as SCL:
   #_w1 := #TRUE AND NOT #statTonTimer[0].Q AND NOT #statTonTimer[1].Q AND "LRemoteAccess_Data".mobilePanel1.ucpPointerDisabled AND ("LRemoteAccess_Data".mobilePanel1.mpKeySwitch <> 0);
   "LRemoteAccess_Data".connectionBoxes[1].connected := #_w1 AND ("LRemoteAccess_Data".connectionBoxes[1].ID = "LRemoteAccess_Data".mobilePanel1.mpReadBoxID);
   "LRemoteAccess_Data".connectionBoxes[2].connected := #_w1 AND ("LRemoteAccess_Data".connectionBoxes[2].ID = "LRemoteAccess_Data".mobilePanel1.mpReadBoxID);
   "LRemoteAccess_Data".mobilePanel1.connectionTerminated := NOT (#TRUE AND NOT #statTonTimer[0].Q AND NOT #statTonTimer[1].Q);
   "Safety.DataToSafety".PhmiCommunicationOK := #TRUE AND NOT "LRemoteAccess_Data".mobilePanel1.connectionTerminated;
   "Safety.DataToSafety".MobilePanelConnected := NOT (#TRUE AND NOT "LRemoteAccess_Data".connectionBoxes[1].connected AND NOT "LRemoteAccess_Data".connectionBoxes[2].connected);
   "Safety.DataToSafety"."PhmiNo1.Connected" := #TRUE AND "LRemoteAccess_Data".connectionBoxes[1].connected;
   "Safety.DataToSafety"."PhmiNo2.Connected" := #TRUE AND "LRemoteAccess_Data".connectionBoxes[2].connected;
   IF #TRUE AND ("LRemoteAccess_Data".mobilePanel1.mpKeySwitch <> 0) THEN
       "Safety.DataToSafety".KeyBoxStatus := 1;
   END_IF;
   IF #TRUE AND ("LRemoteAccess_Data".mobilePanel1.mpKeySwitch = 0) THEN
       "Safety.DataToSafety".KeyBoxStatus := 0;
   END_IF;
END_REGION

REGION Network 14: Connection Box ID Safety Move
   RUNG wire#powerrail
      Move(in := "LRemoteAccess_Data".connectionBoxes[1].ID, out1 => "Safety.DataToSafety".connectionBoxID_1)
      Move(in := "LRemoteAccess_Data".connectionBoxes[2].ID, out1 => "Safety.DataToSafety".connectionBoxID_2)
   END_RUNG
   // the same network as SCL:
   "Safety.DataToSafety".connectionBoxID_1 := "LRemoteAccess_Data".connectionBoxes[1].ID;
   "Safety.DataToSafety".connectionBoxID_2 := "LRemoteAccess_Data".connectionBoxes[2].ID;
END_REGION

REGION Network 15: enable Control Interfaces
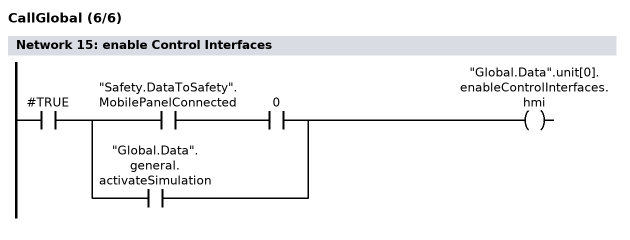
   RUNG wire#powerrail
      Contact( #TRUE )
      wire#w1
      Contact( "Safety.DataToSafety".MobilePanelConnected )
      Contact( 0 )
      wire#w2
      Coil( "Global.Data".unit[0].enableControlInterfaces.hmi )
   END_RUNG
   RUNG wire#w1
      Contact( "Global.Data".general.activateSimulation )
   END_RUNG wire#w2
   // the same network as SCL:
   "Global.Data".unit[0].enableControlInterfaces.hmi := #TRUE AND (("Safety.DataToSafety".MobilePanelConnected AND 0) OR "Global.Data".general.activateSimulation);
END_REGION
END_FUNCTION_BLOCK
